{attribute 'qualified_only'}
VAR_GLOBAL
    Machine            : TMachine;
    Safety             : TSafety;
    HmiInterface       : THmiInterface;
    Logging            : TLogger;
    HydraulicPumpMotor : TMotorStarter;
END_VAR

(* stored: Version 1.1.0.1, ProductVersion 3.1.4024.9
   GVL Objects: Id {7240b198-f5fe-07bb-04a2-7752144c7e95} *)
